(* PLC project v0.6.04_CycleSemiAuto.project, CODESYS CODESYS V3.5 SP19 Patch 1 *)
(* stored: creationDateTime 2026-07-23T22:45:01.538006, modificationDateTime 2026-07-23T22:45:01.538006 *)

(* ═══════════════════════════════════════════════════════════════ 🎮 ST_JoystickCmd — Commandes IHM pour le Joystick ═══════════════════════════════════════════════════════════════ *)
TYPE ST_JoystickCmd : STRUCT
  BtnCalibrate : BOOL;  (* 🎯 Demande de recalage au neutre *)
END_STRUCT;
END_TYPE
